// TIA Portal V17 export
// export: Created 2025-11-19T10:30:00.000Z, ExportSetting WithDefaults, DisplayName Totally Integrated Automation Portal, DisplayVersion V17
FUNCTION "FC_MotorControl" : Void   // FC10, SCL
{ S7_Optimized_Access := 'TRUE' }
AUTHOR : Engineering Team
FAMILY : Motors
NAME : Motor Control Function
VERSION : 1.0
// stored: AutoNumber true, IsIECCheckEnabled true
   VAR_INPUT
      Start : Bool;
      Stop : Bool;
      Speed_Setpoint : Real;
   END_VAR
   VAR_OUTPUT
      Motor_On : Bool;
      Current_Speed : Real;
   END_VAR
   VAR_TEMP
      temp_speed : Real;
   END_VAR
BEGIN
// Motor Control
// Main motor control with speed ramping
   // Motor Control Logic
   IF #Start AND NOT #Stop THEN
       #Motor_On := TRUE;
       #temp_speed := #Speed_Setpoint;

       // Ramp up speed
       IF #Current_Speed < #temp_speed THEN
           #Current_Speed := #Current_Speed + 10.0;
           IF #Current_Speed > #temp_speed THEN
               #Current_Speed := #temp_speed;
           END_IF;
       END_IF;
   ELSE
       #Motor_On := FALSE;
       // Ramp down speed
       IF #Current_Speed > 0.0 THEN
           #Current_Speed := #Current_Speed - 10.0;
           IF #Current_Speed < 0.0 THEN
               #Current_Speed := 0.0;
           END_IF;
       END_IF;
   END_IF;
END_FUNCTION
